(* CODESYS project KickerMotor.xml

Project tree, tasks and I/O mapping:
  function block KickerMotor [LD]
*)

// KickerMotor
FUNCTION_BLOCK KickerMotor
VAR_INPUT
	Forward: 			BOOL;				//
	Brake: 				BOOL;				//
	Settings: 			MotorSettings;		//
END_VAR
VAR_OUTPUT
	MotorOutput: 		BOOL;				//
	BrakeOutput: 		BOOL;				//
END_VAR
VAR
END_VAR

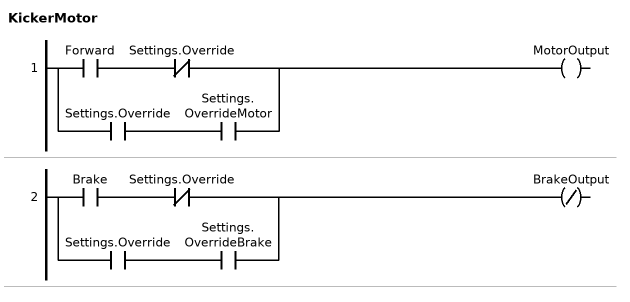
// NETWORK 1
MotorOutput := Forward AND NOT Settings.Override OR Settings.Override AND Settings.OverrideMotor;

// NETWORK 2
BrakeOutput := NOT (Brake AND NOT Settings.Override OR Settings.Override AND Settings.OverrideBrake);

END_FUNCTION_BLOCK
